{attribute 'linkalways'} 
{attribute 'no_explicit_call' := 'This FB is a CLASS and must be accessed using methods or properties'}
{attribute 'enable_dynamic_creation'}
FUNCTION_BLOCK Node_F_VN_MaxElementElementwise_UINT EXTENDS VisionNode
VAR
    ipContainer : _ITcVnContainer;
    nMax : _UINT(0);
    hrPrev : _HRESULT(S_OK);
    hresult : _HRESULT(S_OK);
END_VAR

METHOD PUBLIC  Clone : I_Node
VAR
	pNode : POINTER TO Node_F_VN_MaxElementElementwise_UINT;
END_VAR
pNode := __NEW(Node_F_VN_MaxElementElementwise_UINT);
Clone := pNode^;
END_METHOD

METHOD FB_init : BOOL
VAR_INPUT
	bInitRetains : BOOL; // if TRUE, the retain variables are initialized (warm start / cold start)
	bInCopyCode : BOOL;  // if TRUE, the instance afterwards gets moved into the copy code (online change)
END_VAR
AddInput('ipContainer', ipContainer);
AddInput('nMax', nMax);
AddInput('hrPrev', hrPrev);
AddOutput('ipContainer', ipContainer);
AddOutput('hresult',hresult);
END_METHOD

METHOD PROTECTED OnExecute : HRESULT
hresult.Value := F_VN_MaxElementElementwise_UINT(
    ipContainer := ipContainer.Value,
    nMax := nMax.Value,
    hrPrev:= hrPrev.Value);
END_METHOD

METHOD PUBLIC PreExecutionCheck
VAR_INPUT
	Check : I_PreExecutionChecks;
END_VAR
Check.IsTrue(ipContainer.IsValid, 'ipContainer must be a valid container');
END_METHOD

END_FUNCTION_BLOCK

(* stored: Version 1.1.0.1, ProductVersion 3.1.4024.13
   POU Node_F_VN_MaxElementElementwise_UINT: Id {4201bdab-05b3-41c8-b7e4-458f0a561679}, SpecialFunc None
   Folder Constructor: Id {9b9604ef-9b03-4157-97bb-93e956ee39b4}
   Method Clone: Id {9c82849b-09e8-4ba9-8178-0c5f042d62dd}
   Method FB_init: Id {b6836fdd-df96-4444-a0e1-ba940aa0ad55}
   Method OnExecute: Id {c8daebc1-b6e5-431b-a734-78528c675da6}
   Method PreExecutionCheck: Id {b8c74de6-972c-41c2-b25b-b295290d7158} *)
